# EPICS autosave request: soft_iocs/srs/iocBoot/iocdg645/auto_settings.req
## DG645 digital delay generator settings
file drvDG645_settings.req P=$(P1),R=$(R1)
file drvDG645_settings.req P=$(P2),R=$(R2)
